(* PLC project mqtt, SMARTEH d.o.o. LHC2_GOT_012 1.1.359 *)
(* stored: creationDateTime 2024-07-25T15:43:22, modificationDateTime 2026-08-13T16:02:10 *)

TYPE inner : STRUCT
  a : DINT;
  b : DINT;
  c : STRING;
END_STRUCT;
END_TYPE

TYPE outer : STRUCT
  aa : DINT;
  bb : inner;
  cc : DINT;
END_STRUCT;
END_TYPE

TYPE datatype0 : STRUCT
  kkk : DINT;
  xxx : DINT;
  complex : inner;
END_STRUCT;
END_TYPE

PROGRAM program0
  VAR
    LOGGER0 : LOGGER;
    COUNT : LINT;
  END_VAR
  VAR_EXTERNAL
    MQTT_STATUS_3 : INT;
    MQTT_STATUS_4 : INT;
  END_VAR
  VAR
    json_topic_b_out AT %Q3.0 : datatype0 := (kkk := 1, xxx := 2, complex := (a := 3, b := 4, c := 'a'));  (* mqtt_0/json_topic_b *)
    json_topic_b_in AT %I4.0 : datatype0;  (* mqtt_1/json_topic_b *)
    json_topic_a_in AT %I3.0 : outer;  (* mqtt_0/json_topic_a *)
    json_topic_a_out AT %Q4.0 : outer := (aa := 1, bb := (a := 2, b := 3, c := 'a'), cc := 4);  (* mqtt_1/json_topic_a *)
    dint_topic_b_out AT %QD3.1 : DINT := 42;  (* mqtt_0/dint_topic_b *)
    dint_topic_b_in AT %ID4.1 : DINT;  (* mqtt_1/dint_topic_b *)
    dint_topic_a_in AT %ID3.1 : DINT;  (* mqtt_0/dint_topic_a *)
    dint_topic_a_out AT %QD4.1 : DINT := 117;  (* mqtt_1/dint_topic_a *)
  END_VAR

            (* Simple test checking variables are passed through in both directions *)
IF  (MQTT_STATUS_3 = 1) &
    (MQTT_STATUS_4 = 1) &
    (dint_topic_a_out = dint_topic_a_in) &
    (dint_topic_b_out = dint_topic_b_in) &
    (json_topic_b_out.kkk = json_topic_b_in.kkk) &
    (json_topic_b_out.xxx = json_topic_b_in.xxx) &
    (json_topic_b_out.complex.a = json_topic_b_in.complex.a) &
    (json_topic_b_out.complex.b = json_topic_b_in.complex.b) &
    (json_topic_b_out.complex.c = json_topic_b_in.complex.c) &
    (json_topic_a_out.aa = json_topic_a_in.aa) &
    (json_topic_a_out.bb.a = json_topic_a_in.bb.a) &
    (json_topic_a_out.bb.b = json_topic_a_in.bb.b) &
    (json_topic_a_out.bb.c = json_topic_a_in.bb.c) &
    (json_topic_a_out.cc = json_topic_a_in.cc) THEN
  LOGGER0(
     TRIG := TRUE,
     MSG := 'TEST OK',
     LEVEL := CRITICAL);

END_IF;
COUNT:=COUNT+1;

          
END_PROGRAM

CONFIGURATION config
  VAR_GLOBAL
    GlobalVar0 : datatype0;
  END_VAR
  RESOURCE resource1 ON PLC
    TASK main_task(INTERVAL := T#1000ms, PRIORITY := 0);
    PROGRAM instance0 WITH main_task : program0;
  END_RESOURCE
END_CONFIGURATION
